TYPE ST_UninitializedStartUpFrame :
STRUCT
	iProgressBar					: USINT;
	bCR800EtherCatInitialization	: BOOL;
END_STRUCT
END_TYPE

(* stored: Version 1.1.0.1, ProductVersion 3.1.4024.9
   DUT ST_UninitializedStartUpFrame: Id {8a512a69-219a-45d2-9de8-50ae40df44da} *)
